{attribute 'qualified_only'}
{attribute 'strict'}
TYPE e_StatoWorkOrder :
(
	NON_ESEGUITO 	:= 0,
	DA_ESEGUIRE		:= 1,
	IN_ESECUZIONE 	:= 2,
	TERMINATO		:= 3
);
END_TYPE

(* stored: Version 1.1.0.1, ProductVersion 3.1.4024.11
   DUT e_StatoWorkOrder: Id {667882e8-04dc-4fba-8c8f-d6593b58ba84} *)
